TYPE "TMeasuringCtrl"
VERSION : 0.1
// Block: TMeasuringCtrl
   STRUCT
      Rst : Bool;
      MeasureEnable : Bool;
      Mode : DInt;
   END_STRUCT;

END_TYPE
